  MoveL 4411 to (296.71, 215.61, -10) mm, rotated rx -180 ry 0 rz 180 deg; joints [-8.145, -42.25, 106.462, 170.968, 64.491, -176.084]
  MoveL 4412 to (298.79, 218.64, -10) mm, rotated rx 180 ry 0 rz 180 deg; joints [-8.247, -42.193, 106.293, 170.847, 64.387, -176.016]
  MoveL 4413 to (300.68, 221.8, -10) mm, rotated rx 180 ry 0 rz 180 deg; joints [-8.354, -42.14, 106.135, 170.72, 64.292, -175.946]
  MoveL 4414 to (302.37, 225.07, -10) mm, rotated rx -180 ry 0 rz -180 deg; joints [-8.466, -42.091, 105.99, 170.589, 64.205, -175.874]
  MoveL 4415 to (303.85, 228.44, -10) mm, rotated rx -180 ry 0 rz 180 deg; joints [-8.583, -42.046, 105.857, 170.452, 64.127, -175.802]
  MoveL 4416 to (305.1, 231.9, -10) mm, rotated rx -180 ry 0 rz -180 deg; joints [-8.704, -42.005, 105.737, 170.312, 64.058, -175.729]
  MoveL 4417 to (306.14, 235.43, -10) mm, rotated rx 180 ry 0 rz 180 deg; joints [-8.828, -41.969, 105.631, 170.168, 63.998, -175.655]
  MoveL 4418 to (306.95, 239.02, -10) mm, rotated rx 180 ry 0 rz -180 deg; joints [-8.956, -41.937, 105.539, 170.021, 63.948, -175.581]
  MoveL 4419 to (307.53, 242.66, -10) mm, rotated rx -180 ry 0 rz 180 deg; joints [-9.087, -41.911, 105.461, 169.872, 63.908, -175.508]
  MoveL 4420 to (307.88, 246.32, -10) mm, rotated rx -180 ry 0 rz -180 deg; joints [-9.219, -41.889, 105.398, 169.721, 63.877, -175.435]
  MoveL 4421 to (308, 250, -10) mm, rotated rx 180 ry 0 rz 180 deg; joints [-9.354, -41.873, 105.35, 169.569, 63.857, -175.363]
  MoveL 4422 to (296, 250, -10) mm, rotated rx 180 ry 0 rz 180 deg; joints [-9.427, -42.146, 106.154, 169.534, 64.384, -175.434]
  MoveL 4423 to (295.91, 252.92, -10) mm, rotated rx -180 ry 0 rz 180 deg; joints [-9.536, -42.137, 106.127, 169.413, 64.376, -175.379]
  MoveL 4424 to (295.63, 255.82, -10) mm, rotated rx -180 ry 0 rz 180 deg; joints [-9.645, -42.132, 106.113, 169.291, 64.375, -175.324]
  MoveL 4425 to (295.17, 258.71, -10) mm, rotated rx -180 ry 0 rz -180 deg; joints [-9.755, -42.132, 106.111, 169.17, 64.383, -175.272]
  MoveL 4426 to (294.53, 261.55, -10) mm, rotated rx -180 ry 0 rz 180 deg; joints [-9.864, -42.135, 106.121, 169.05, 64.399, -175.221]
  MoveL 4427 to (293.7, 264.35, -10) mm, rotated rx 180 ry 0 rz 180 deg; joints [-9.973, -42.142, 106.143, 168.931, 64.422, -175.172]
  MoveL 4428 to (292.7, 267.1, -10) mm, rotated rx 180 ry 0 rz 180 deg; joints [-10.081, -42.154, 106.177, 168.814, 64.453, -175.125]
  MoveL 4429 to (291.53, 269.77, -10) mm, rotated rx 180 ry 0 rz 180 deg; joints [-10.187, -42.17, 106.223, 168.699, 64.493, -175.081]
  MoveL 4430 to (290.2, 272.37, -10) mm, rotated rx -180 ry 0 rz -180 deg; joints [-10.292, -42.189, 106.281, 168.587, 64.539, -175.04]
  MoveL 4431 to (288.7, 274.87, -10) mm, rotated rx 180 ry 0 rz 180 deg; joints [-10.395, -42.213, 106.351, 168.478, 64.593, -175.001]
  MoveL 4432 to (287.04, 277.27, -10) mm, rotated rx 180 ry 0 rz 180 deg; joints [-10.495, -42.24, 106.431, 168.372, 64.654, -174.966]
  MoveL 4433 to (285.24, 279.57, -10) mm, rotated rx 180 ry 0 rz 180 deg; joints [-10.593, -42.271, 106.523, 168.271, 64.722, -174.934]
  MoveL 4434 to (283.29, 281.74, -10) mm, rotated rx 180 ry 0 rz -180 deg; joints [-10.687, -42.305, 106.625, 168.174, 64.797, -174.905]
  MoveL 4435 to (281.21, 283.79, -10) mm, rotated rx -180 ry 0 rz -180 deg; joints [-10.777, -42.342, 106.737, 168.081, 64.878, -174.879]
  MoveL 4436 to (279.01, 285.7, -10) mm, rotated rx 180 ry 0 rz -180 deg; joints [-10.864, -42.383, 106.859, 167.994, 64.965, -174.857]
  MoveL 4437 to (276.68, 287.47, -10) mm, rotated rx 180 ry 0 rz 180 deg; joints [-10.946, -42.427, 106.99, 167.912, 65.058, -174.839]
  MoveL 4438 to (274.25, 289.09, -10) mm, rotated rx -180 ry 0 rz -180 deg; joints [-11.024, -42.474, 107.13, 167.836, 65.156, -174.825]
  MoveL 4439 to (271.72, 290.55, -10) mm, rotated rx 180 ry 0 rz -180 deg; joints [-11.096, -42.523, 107.278, 167.766, 65.259, -174.815]
  MoveL 4440 to (269.11, 291.84, -10) mm, rotated rx 180 ry 0 rz -180 deg; joints [-11.164, -42.575, 107.433, 167.702, 65.366, -174.808]
  MoveL 4441 to (266.42, 292.97, -10) mm, rotated rx -180 ry 0 rz -180 deg; joints [-11.226, -42.629, 107.596, 167.644, 65.478, -174.805]
  MoveL 4442 to (263.66, 293.93, -10) mm, rotated rx -180 ry 0 rz -180 deg; joints [-11.282, -42.685, 107.765, 167.594, 65.594, -174.806]
  MoveL 4443 to (260.84, 294.7, -10) mm, rotated rx -180 ry 0 rz -180 deg; joints [-11.332, -42.742, 107.939, 167.551, 65.712, -174.811]
  MoveL 4444 to (257.99, 295.3, -10) mm, rotated rx -180 ry 0 rz 180 deg; joints [-11.376, -42.801, 108.119, 167.514, 65.834, -174.82]
  MoveL 4445 to (255.1, 295.72, -10) mm, rotated rx -180 ry 0 rz -180 deg; joints [-11.414, -42.861, 108.303, 167.485, 65.958, -174.833]
  MoveL 4446 to (252.19, 295.95, -10) mm, rotated rx 180 ry 0 rz -180 deg; joints [-11.444, -42.923, 108.49, 167.464, 66.084, -174.849]
  MoveL 4447 to (249.27, 295.99, -10) mm, rotated rx 180 ry 0 rz 180 deg; joints [-11.468, -42.985, 108.68, 167.45, 66.211, -174.869]
  MoveL 4448 to (246.35, 295.86, -10) mm, rotated rx 180 ry 0 rz -180 deg; joints [-11.486, -43.047, 108.872, 167.444, 66.339, -174.892]
  MoveL 4449 to (243.45, 295.53, -10) mm, rotated rx 180 ry 0 rz -180 deg; joints [-11.496, -43.11, 109.065, 167.445, 66.467, -174.919]
  MoveL 4450 to (240.58, 295.02, -10) mm, rotated rx -180 ry 0 rz -180 deg; joints [-11.499, -43.172, 109.259, 167.454, 66.596, -174.949]
  MoveL 4451 to (237.74, 294.34, -10) mm, rotated rx 180 ry 0 rz 180 deg; joints [-11.494, -43.234, 109.452, 167.471, 66.723, -174.981]
  MoveL 4452 to (234.95, 293.47, -10) mm, rotated rx -180 ry 0 rz -180 deg; joints [-11.483, -43.296, 109.645, 167.496, 66.85, -175.017]
  MoveL 4453 to (232.23, 292.43, -10) mm, rotated rx 180 ry 0 rz -180 deg; joints [-11.464, -43.357, 109.835, 167.528, 66.975, -175.056]
  MoveL 4454 to (229.57, 291.22, -10) mm, rotated rx -180 ry 0 rz 180 deg; joints [-11.439, -43.417, 110.023, 167.568, 67.098, -175.096]
  MoveL 4455 to (227, 289.84, -10) mm, rotated rx -180 ry 0 rz -180 deg; joints [-11.406, -43.475, 110.207, 167.615, 67.218, -175.14]
  MoveL 4456 to (224.52, 288.3, -10) mm, rotated rx 180 ry 0 rz 180 deg; joints [-11.366, -43.532, 110.388, 167.669, 67.335, -175.185]
  MoveL 4457 to (222.14, 286.6, -10) mm, rotated rx -180 ry 0 rz -180 deg; joints [-11.319, -43.588, 110.563, 167.73, 67.448, -175.232]
  MoveL 4458 to (219.88, 284.76, -10) mm, rotated rx 180 ry 0 rz -180 deg; joints [-11.266, -43.641, 110.733, 167.798, 67.558, -175.281]
  MoveL 4459 to (217.73, 282.78, -10) mm, rotated rx -180 ry 0 rz -180 deg; joints [-11.206, -43.692, 110.897, 167.872, 67.663, -175.331]
  MoveL 4460 to (215.72, 280.67, -10) mm, rotated rx 180 ry 0 rz 180 deg; joints [-11.139, -43.741, 111.053, 167.953, 67.762, -175.382]
  MoveL 4461 to (213.84, 278.44, -10) mm, rotated rx 180 ry 0 rz -180 deg; joints [-11.067, -43.788, 111.202, 168.039, 67.857, -175.435]
  MoveL 4462 to (212.11, 276.08, -10) mm, rotated rx -180 ry 0 rz -180 deg; joints [-10.989, -43.832, 111.343, 168.131, 67.946, -175.488]
  MoveL 4463 to (210.53, 273.63, -10) mm, rotated rx -180 ry 0 rz -180 deg; joints [-10.905, -43.873, 111.475, 168.229, 68.028, -175.542]
  MoveL 4464 to (209.11, 271.08, -10) mm, rotated rx 180 ry 0 rz 180 deg; joints [-10.817, -43.91, 111.598, 168.331, 68.104, -175.596]
  MoveL 4465 to (207.86, 268.44, -10) mm, rotated rx -180 ry 0 rz -180 deg; joints [-10.723, -43.945, 111.71, 168.438, 68.174, -175.65]
  MoveL 4466 to (206.77, 265.73, -10) mm, rotated rx 180 ry 0 rz -180 deg; joints [-10.625, -43.977, 111.813, 168.549, 68.236, -175.705]
  MoveL 4467 to (205.86, 262.96, -10) mm, rotated rx 180 ry 0 rz -180 deg; joints [-10.523, -44.005, 111.905, 168.663, 68.29, -175.759]
  MoveL 4468 to (205.13, 260.13, -10) mm, rotated rx 180 ry 0 rz -180 deg; joints [-10.418, -44.03, 111.985, 168.78, 68.337, -175.812]
  MoveL 4469 to (204.58, 257.27, -10) mm, rotated rx 180 ry 0 rz 180 deg; joints [-10.31, -44.051, 112.054, 168.9, 68.377, -175.865]
  MoveL 4470 to (204.21, 254.37, -10) mm, rotated rx -180 ry 0 rz 180 deg; joints [-10.199, -44.068, 112.112, 169.022, 68.408, -175.917]
  MoveL 4471 to (204.02, 251.46, -10) mm, rotated rx 180 ry 0 rz 180 deg; joints [-10.086, -44.082, 112.157, 169.146, 68.431, -175.968]
  MoveL 4472 to (204.02, 248.54, -10) mm, rotated rx 180 ry 0 rz 180 deg; joints [-9.971, -44.092, 112.19, 169.271, 68.445, -176.018]
  MoveL 4473 to (204.21, 245.63, -10) mm, rotated rx 180 ry 0 rz -180 deg; joints [-9.855, -44.099, 112.211, 169.396, 68.451, -176.066]
  MoveL 4474 to (204.58, 242.73, -10) mm, rotated rx 180 ry 0 rz -180 deg; joints [-9.739, -44.101, 112.219, 169.521, 68.449, -176.113]
  MoveL 4475 to (205.13, 239.87, -10) mm, rotated rx 180 ry 0 rz -180 deg; joints [-9.622, -44.1, 112.215, 169.646, 68.439, -176.159]
  MoveL 4476 to (205.86, 237.04, -10) mm, rotated rx 180 ry 0 rz 180 deg; joints [-9.506, -44.095, 112.199, 169.77, 68.42, -176.202]
  MoveL 4477 to (206.77, 234.27, -10) mm, rotated rx -180 ry 0 rz 180 deg; joints [-9.391, -44.086, 112.17, 169.892, 68.392, -176.244]
  MoveL 4478 to (207.86, 231.56, -10) mm, rotated rx -180 ry 0 rz -180 deg; joints [-9.277, -44.074, 112.129, 170.012, 68.357, -176.284]
  MoveL 4479 to (209.11, 228.92, -10) mm, rotated rx 180 ry 0 rz 180 deg; joints [-9.166, -44.057, 112.075, 170.13, 68.313, -176.321]
  MoveL 4480 to (210.53, 226.37, -10) mm, rotated rx 180 ry 0 rz -180 deg; joints [-9.056, -44.037, 112.01, 170.244, 68.262, -176.356]
  MoveL 4481 to (212.11, 223.92, -10) mm, rotated rx -180 ry 0 rz 180 deg; joints [-8.95, -44.014, 111.934, 170.355, 68.202, -176.389]
  MoveL 4482 to (213.84, 221.56, -10) mm, rotated rx 180 ry 0 rz 180 deg; joints [-8.847, -43.987, 111.846, 170.461, 68.136, -176.419]
  MoveL 4483 to (215.72, 219.33, -10) mm, rotated rx -180 ry 0 rz 180 deg; joints [-8.747, -43.957, 111.747, 170.564, 68.062, -176.447]
  MoveL 4484 to (217.73, 217.22, -10) mm, rotated rx -180 ry 0 rz 180 deg; joints [-8.652, -43.923, 111.638, 170.661, 67.982, -176.472]
  MoveL 4485 to (219.88, 215.24, -10) mm, rotated rx 180 ry 0 rz 180 deg; joints [-8.562, -43.886, 111.518, 170.753, 67.895, -176.494]
  MoveL 4486 to (222.14, 213.4, -10) mm, rotated rx 180 ry 0 rz -180 deg; joints [-8.477, -43.846, 111.39, 170.839, 67.802, -176.513]
  MoveL 4487 to (224.52, 211.7, -10) mm, rotated rx 180 ry 0 rz -180 deg; joints [-8.397, -43.803, 111.252, 170.919, 67.703, -176.53]
  MoveL 4488 to (227, 210.16, -10) mm, rotated rx -180 ry 0 rz 180 deg; joints [-8.322, -43.758, 111.106, 170.993, 67.599, -176.543]
  MoveL 4489 to (229.57, 208.78, -10) mm, rotated rx 180 ry 0 rz -180 deg; joints [-8.254, -43.71, 110.952, 171.06, 67.491, -176.554]
  MoveL 4490 to (232.23, 207.57, -10) mm, rotated rx 180 ry 0 rz -180 deg; joints [-8.192, -43.659, 110.79, 171.12, 67.378, -176.561]
  MoveL 4491 to (234.95, 206.53, -10) mm, rotated rx 180 ry 0 rz 180 deg; joints [-8.136, -43.606, 110.623, 171.173, 67.261, -176.565]
  MoveL 4492 to (237.74, 205.66, -10) mm, rotated rx -180 ry 0 rz -180 deg; joints [-8.087, -43.552, 110.449, 171.219, 67.14, -176.566]
  MoveL 4493 to (240.58, 204.98, -10) mm, rotated rx -180 ry 0 rz -180 deg; joints [-8.045, -43.495, 110.27, 171.257, 67.017, -176.563]
  MoveL 4494 to (243.45, 204.47, -10) mm, rotated rx 180 ry 0 rz 180 deg; joints [-8.009, -43.437, 110.087, 171.287, 66.891, -176.558]
  MoveL 4495 to (246.35, 204.14, -10) mm, rotated rx -180 ry 0 rz 180 deg; joints [-7.981, -43.378, 109.9, 171.309, 66.763, -176.549]
  MoveL 4496 to (249.27, 204.01, -10) mm, rotated rx -180 ry 0 rz -180 deg; joints [-7.96, -43.317, 109.711, 171.324, 66.635, -176.537]
  MoveL 4497 to (252.19, 204.05, -10) mm, rotated rx 180 ry 0 rz -180 deg; joints [-7.946, -43.256, 109.519, 171.33, 66.505, -176.521]
  MoveL 4498 to (255.1, 204.28, -10) mm, rotated rx -180 ry 0 rz -180 deg; joints [-7.939, -43.194, 109.326, 171.329, 66.375, -176.503]
  MoveL 4499 to (257.99, 204.7, -10) mm, rotated rx 180 ry 0 rz 180 deg; joints [-7.94, -43.131, 109.132, 171.32, 66.245, -176.481]
  MoveL 4500 to (260.84, 205.3, -10) mm, rotated rx 180 ry 0 rz 180 deg; joints [-7.947, -43.069, 108.938, 171.303, 66.116, -176.456]
  MoveL 4501 to (263.66, 206.07, -10) mm, rotated rx -180 ry 0 rz -180 deg; joints [-7.962, -43.006, 108.746, 171.278, 65.989, -176.428]
  MoveL 4502 to (266.42, 207.03, -10) mm, rotated rx -180 ry 0 rz -180 deg; joints [-7.984, -42.944, 108.555, 171.246, 65.863, -176.397]
  MoveL 4503 to (269.11, 208.16, -10) mm, rotated rx 180 ry 0 rz 180 deg; joints [-8.012, -42.882, 108.367, 171.206, 65.739, -176.363]
  MoveL 4504 to (271.72, 209.45, -10) mm, rotated rx -180 ry 0 rz -180 deg; joints [-8.047, -42.822, 108.182, 171.159, 65.619, -176.326]
  MoveL 4505 to (274.25, 210.91, -10) mm, rotated rx -180 ry 0 rz -180 deg; joints [-8.089, -42.762, 108.001, 171.104, 65.501, -176.286]
  MoveL 4506 to (276.68, 212.53, -10) mm, rotated rx 180 ry 0 rz -180 deg; joints [-8.137, -42.704, 107.824, 171.043, 65.387, -176.244]
  MoveL 4507 to (279.01, 214.3, -10) mm, rotated rx 180 ry 0 rz -180 deg; joints [-8.191, -42.648, 107.654, 170.976, 65.278, -176.2]
  MoveL 4508 to (281.21, 216.21, -10) mm, rotated rx -180 ry 0 rz 180 deg; joints [-8.251, -42.593, 107.489, 170.902, 65.173, -176.153]
  MoveL 4509 to (283.29, 218.26, -10) mm, rotated rx 180 ry 0 rz 180 deg; joints [-8.317, -42.541, 107.331, 170.822, 65.073, -176.104]
  MoveL 4510 to (285.24, 220.43, -10) mm, rotated rx 180 ry 0 rz -180 deg; joints [-8.388, -42.491, 107.18, 170.736, 64.979, -176.054]
  MoveL 4511 to (287.04, 222.73, -10) mm, rotated rx 180 ry 0 rz 180 deg; joints [-8.464, -42.443, 107.037, 170.645, 64.89, -176.001]
  MoveL 4512 to (288.7, 225.13, -10) mm, rotated rx 180 ry 0 rz -180 deg; joints [-8.545, -42.398, 106.903, 170.549, 64.808, -175.947]
  MoveL 4513 to (290.2, 227.64, -10) mm, rotated rx -180 ry 0 rz -180 deg; joints [-8.63, -42.356, 106.778, 170.449, 64.732, -175.892]
  MoveL 4514 to (291.53, 230.23, -10) mm, rotated rx 180 ry 0 rz 180 deg; joints [-8.719, -42.317, 106.662, 170.345, 64.663, -175.836]
  MoveL 4515 to (292.7, 232.9, -10) mm, rotated rx 180 ry 0 rz 180 deg; joints [-8.812, -42.282, 106.557, 170.236, 64.6, -175.779]
  MoveL 4516 to (293.7, 235.65, -10) mm, rotated rx -180 ry 0 rz -180 deg; joints [-8.908, -42.25, 106.462, 170.125, 64.545, -175.721]
  MoveL 4517 to (294.53, 238.45, -10) mm, rotated rx -180 ry 0 rz -180 deg; joints [-9.007, -42.222, 106.377, 170.011, 64.497, -175.663]
  MoveL 4518 to (295.17, 241.29, -10) mm, rotated rx -180 ry 0 rz -180 deg; joints [-9.109, -42.197, 106.304, 169.894, 64.457, -175.605]
  MoveL 4519 to (295.63, 244.18, -10) mm, rotated rx 180 ry 0 rz 180 deg; joints [-9.214, -42.176, 106.242, 169.775, 64.425, -175.548]
  MoveL 4520 to (295.91, 247.08, -10) mm, rotated rx -180 ry 0 rz -180 deg; joints [-9.32, -42.159, 106.192, 169.655, 64.401, -175.49]
  MoveL 4521 to (296, 250, -10) mm, rotated rx 180 ry 0 rz 180 deg; joints [-9.427, -42.146, 106.154, 169.534, 64.384, -175.434]
  MoveL 4522 to (284, 250, -10) mm, rotated rx -180 ry 0 rz 180 deg; joints [-9.502, -42.415, 106.953, 169.498, 64.912, -175.506]
  MoveL 4523 to (283.93, 252.16, -10) mm, rotated rx 180 ry 0 rz -180 deg; joints [-9.582, -42.408, 106.933, 169.408, 64.905, -175.465]
  MoveL 4524 to (283.73, 254.3, -10) mm, rotated rx -180 ry 0 rz 180 deg; joints [-9.664, -42.405, 106.923, 169.318, 64.905, -175.426]
  MoveL 4525 to (283.39, 256.43, -10) mm, rotated rx 180 ry 0 rz -180 deg; joints [-9.745, -42.404, 106.921, 169.228, 64.91, -175.388]
  MoveL 4526 to (282.91, 258.54, -10) mm, rotated rx 180 ry 0 rz 180 deg; joints [-9.827, -42.407, 106.929, 169.139, 64.922, -175.351]
  MoveL 4527 to (282.3, 260.61, -10) mm, rotated rx 180 ry 0 rz -180 deg; joints [-9.908, -42.412, 106.945, 169.05, 64.939, -175.315]
  MoveL 4528 to (281.56, 262.64, -10) mm, rotated rx 180 ry 0 rz 180 deg; joints [-9.988, -42.421, 106.971, 168.963, 64.962, -175.281]
  MoveL 4529 to (280.7, 264.61, -10) mm, rotated rx 180 ry 0 rz 180 deg; joints [-10.068, -42.432, 107.005, 168.878, 64.991, -175.249]
  MoveL 4530 to (279.71, 266.53, -10) mm, rotated rx 180 ry 0 rz 180 deg; joints [-10.146, -42.446, 107.048, 168.795, 65.026, -175.219]
  MoveL 4531 to (278.6, 268.38, -10) mm, rotated rx 180 ry 0 rz 180 deg; joints [-10.222, -42.464, 107.099, 168.714, 65.066, -175.191]
  MoveL 4532 to (277.38, 270.16, -10) mm, rotated rx -180 ry 0 rz -180 deg; joints [-10.297, -42.483, 107.159, 168.636, 65.111, -175.165]
  MoveL 4533 to (276.05, 271.85, -10) mm, rotated rx 180 ry 0 rz -180 deg; joints [-10.369, -42.506, 107.226, 168.56, 65.161, -175.141]
  MoveL 4534 to (274.61, 273.46, -10) mm, rotated rx 180 ry 0 rz 180 deg; joints [-10.439, -42.531, 107.302, 168.488, 65.217, -175.12]
  MoveL 4535 to (273.07, 274.98, -10) mm, rotated rx 180 ry 0 rz 180 deg; joints [-10.506, -42.559, 107.385, 168.42, 65.277, -175.102]
  MoveL 4536 to (271.44, 276.39, -10) mm, rotated rx -180 ry 0 rz 180 deg; joints [-10.57, -42.589, 107.475, 168.355, 65.341, -175.086]
  MoveL 4537 to (269.72, 277.7, -10) mm, rotated rx 180 ry 0 rz 180 deg; joints [-10.631, -42.621, 107.572, 168.294, 65.41, -175.072]
  MoveL 4538 to (267.93, 278.89, -10) mm, rotated rx 180 ry 0 rz 180 deg; joints [-10.688, -42.655, 107.676, 168.238, 65.483, -175.062]
  MoveL 4539 to (266.06, 279.97, -10) mm, rotated rx 180 ry 0 rz 180 deg; joints [-10.742, -42.691, 107.786, 168.186, 65.56, -175.054]
  MoveL 4540 to (264.12, 280.93, -10) mm, rotated rx 180 ry 0 rz -180 deg; joints [-10.792, -42.729, 107.901, 168.139, 65.639, -175.049]
  MoveL 4541 to (262.13, 281.76, -10) mm, rotated rx 180 ry 0 rz 180 deg; joints [-10.837, -42.769, 108.021, 168.097, 65.722, -175.047]
  MoveL 4542 to (260.1, 282.47, -10) mm, rotated rx 180 ry 0 rz -180 deg; joints [-10.879, -42.81, 108.146, 168.059, 65.808, -175.047]
  MoveL 4543 to (258.02, 283.04, -10) mm, rotated rx -180 ry 0 rz -180 deg; joints [-10.915, -42.852, 108.275, 168.027, 65.896, -175.05]
  MoveL 4544 to (255.9, 283.48, -10) mm, rotated rx 180 ry 0 rz -180 deg; joints [-10.947, -42.896, 108.408, 168.001, 65.986, -175.056]
  MoveL 4545 to (253.77, 283.79, -10) mm, rotated rx -180 ry 0 rz 180 deg; joints [-10.974, -42.94, 108.544, 167.98, 66.078, -175.065]
  MoveL 4546 to (251.62, 283.96, -10) mm, rotated rx 180 ry 0 rz -180 deg; joints [-10.997, -42.985, 108.683, 167.964, 66.171, -175.077]
  MoveL 4547 to (249.46, 284, -10) mm, rotated rx 180 ry 0 rz -180 deg; joints [-11.014, -43.031, 108.823, 167.954, 66.266, -175.091]
  MoveL 4548 to (247.31, 283.89, -10) mm, rotated rx -180 ry 0 rz -180 deg; joints [-11.026, -43.077, 108.965, 167.95, 66.36, -175.107]
  MoveL 4549 to (245.16, 283.65, -10) mm, rotated rx -180 ry 0 rz 180 deg; joints [-11.033, -43.123, 109.108, 167.951, 66.456, -175.127]
  MoveL 4550 to (243.04, 283.28, -10) mm, rotated rx 180 ry 0 rz 180 deg; joints [-11.034, -43.17, 109.251, 167.958, 66.551, -175.148]
  MoveL 4551 to (240.94, 282.77, -10) mm, rotated rx -180 ry 0 rz 180 deg; joints [-11.03, -43.216, 109.394, 167.971, 66.645, -175.172]
  MoveL 4552 to (238.88, 282.13, -10) mm, rotated rx 180 ry 0 rz -180 deg; joints [-11.021, -43.261, 109.536, 167.99, 66.739, -175.197]
  MoveL 4553 to (236.86, 281.36, -10) mm, rotated rx -180 ry 0 rz -180 deg; joints [-11.007, -43.306, 109.677, 168.014, 66.831, -175.225]
  MoveL 4554 to (234.9, 280.46, -10) mm, rotated rx -180 ry 0 rz -180 deg; joints [-10.987, -43.351, 109.816, 168.044, 66.922, -175.255]
  MoveL 4555 to (233, 279.44, -10) mm, rotated rx 180 ry 0 rz -180 deg; joints [-10.962, -43.394, 109.952, 168.079, 67.01, -175.286]
  MoveL 4556 to (231.17, 278.31, -10) mm, rotated rx 180 ry 0 rz -180 deg; joints [-10.932, -43.437, 110.085, 168.119, 67.097, -175.319]
  MoveL 4557 to (229.41, 277.06, -10) mm, rotated rx 180 ry 0 rz 180 deg; joints [-10.897, -43.478, 110.215, 168.165, 67.18, -175.354]
  MoveL 4558 to (227.73, 275.7, -10) mm, rotated rx -180 ry 0 rz 180 deg; joints [-10.857, -43.517, 110.34, 168.215, 67.261, -175.389]
  MoveL 4559 to (226.15, 274.23, -10) mm, rotated rx 180 ry 0 rz 180 deg; joints [-10.813, -43.555, 110.461, 168.27, 67.338, -175.426]
  MoveL 4560 to (224.66, 272.67, -10) mm, rotated rx 180 ry 0 rz -180 deg; joints [-10.763, -43.592, 110.576, 168.33, 67.412, -175.464]
  MoveL 4561 to (223.27, 271.02, -10) mm, rotated rx -180 ry 0 rz -180 deg; joints [-10.71, -43.626, 110.686, 168.394, 67.481, -175.503]
  MoveL 4562 to (221.99, 269.28, -10) mm, rotated rx 180 ry 0 rz -180 deg; joints [-10.652, -43.659, 110.79, 168.463, 67.547, -175.542]
  MoveL 4563 to (220.83, 267.46, -10) mm, rotated rx -180 ry 0 rz 180 deg; joints [-10.59, -43.69, 110.887, 168.535, 67.607, -175.582]
  MoveL 4564 to (219.78, 265.58, -10) mm, rotated rx -180 ry 0 rz -180 deg; joints [-10.525, -43.718, 110.978, 168.61, 67.663, -175.622]
  MoveL 4565 to (218.85, 263.63, -10) mm, rotated rx 180 ry 0 rz 180 deg; joints [-10.456, -43.744, 111.061, 168.689, 67.714, -175.662]
  MoveL 4566 to (218.05, 261.63, -10) mm, rotated rx -180 ry 0 rz -180 deg; joints [-10.384, -43.767, 111.136, 168.771, 67.76, -175.703]
  MoveL 4567 to (217.38, 259.58, -10) mm, rotated rx -180 ry 0 rz -180 deg; joints [-10.309, -43.788, 111.204, 168.855, 67.8, -175.743]
  MoveL 4568 to (216.84, 257.49, -10) mm, rotated rx -180 ry 0 rz -180 deg; joints [-10.232, -43.807, 111.263, 168.942, 67.834, -175.783]
  MoveL 4569 to (216.43, 255.37, -10) mm, rotated rx 180 ry 0 rz 180 deg; joints [-10.152, -43.823, 111.314, 169.03, 67.863, -175.822]
  MoveL 4570 to (216.15, 253.23, -10) mm, rotated rx 180 ry 0 rz -180 deg; joints [-10.071, -43.836, 111.356, 169.12, 67.885, -175.861]
  MoveL 4571 to (216.02, 251.08, -10) mm, rotated rx -180 ry 0 rz -180 deg; joints [-9.988, -43.846, 111.39, 169.211, 67.902, -175.9]
  MoveL 4572 to (216.02, 248.92, -10) mm, rotated rx -180 ry 0 rz 180 deg; joints [-9.904, -43.854, 111.414, 169.303, 67.913, -175.937]
  MoveL 4573 to (216.15, 246.77, -10) mm, rotated rx -180 ry 0 rz 180 deg; joints [-9.819, -43.858, 111.429, 169.395, 67.917, -175.974]
  MoveL 4574 to (216.43, 244.63, -10) mm, rotated rx 180 ry 0 rz -180 deg; joints [-9.733, -43.86, 111.436, 169.487, 67.915, -176.009]
  MoveL 4575 to (216.84, 242.51, -10) mm, rotated rx -180 ry 0 rz 180 deg; joints [-9.648, -43.859, 111.433, 169.579, 67.907, -176.043]
  MoveL 4576 to (217.38, 240.42, -10) mm, rotated rx -180 ry 0 rz -180 deg; joints [-9.563, -43.856, 111.42, 169.67, 67.893, -176.076]
  MoveL 4577 to (218.05, 238.37, -10) mm, rotated rx -180 ry 0 rz -180 deg; joints [-9.478, -43.849, 111.399, 169.76, 67.873, -176.107]
  MoveL 4578 to (218.85, 236.37, -10) mm, rotated rx 180 ry 0 rz 180 deg; joints [-9.395, -43.84, 111.369, 169.848, 67.847, -176.137]
  MoveL 4579 to (219.78, 234.42, -10) mm, rotated rx 180 ry 0 rz -180 deg; joints [-9.313, -43.827, 111.33, 169.935, 67.815, -176.166]
  MoveL 4580 to (220.83, 232.53, -10) mm, rotated rx -180 ry 0 rz 180 deg; joints [-9.233, -43.813, 111.282, 170.019, 67.777, -176.192]
  MoveL 4581 to (221.99, 230.72, -10) mm, rotated rx 180 ry 0 rz -180 deg; joints [-9.155, -43.795, 111.225, 170.101, 67.733, -176.217]
  MoveL 4582 to (223.27, 228.98, -10) mm, rotated rx -180 ry 0 rz 180 deg; joints [-9.079, -43.775, 111.16, 170.179, 67.684, -176.239]
  MoveL 4583 to (224.66, 227.33, -10) mm, rotated rx -180 ry 0 rz 180 deg; joints [-9.006, -43.752, 111.088, 170.254, 67.63, -176.26]
  MoveL 4584 to (226.15, 225.77, -10) mm, rotated rx -180 ry 0 rz 180 deg; joints [-8.936, -43.727, 111.007, 170.326, 67.571, -176.279]
  MoveL 4585 to (227.73, 224.3, -10) mm, rotated rx -180 ry 0 rz 180 deg; joints [-8.869, -43.7, 110.919, 170.394, 67.507, -176.295]
  MoveL 4586 to (229.41, 222.94, -10) mm, rotated rx 180 ry 0 rz 180 deg; joints [-8.806, -43.67, 110.824, 170.458, 67.439, -176.31]
  MoveL 4587 to (231.17, 221.69, -10) mm, rotated rx -180 ry 0 rz 180 deg; joints [-8.747, -43.638, 110.723, 170.517, 67.366, -176.322]
  MoveL 4588 to (233, 220.56, -10) mm, rotated rx 180 ry 0 rz -180 deg; joints [-8.692, -43.604, 110.615, 170.571, 67.29, -176.332]
  MoveL 4589 to (234.9, 219.54, -10) mm, rotated rx 180 ry 0 rz -180 deg; joints [-8.641, -43.568, 110.501, 170.621, 67.21, -176.339]
  MoveL 4590 to (236.86, 218.64, -10) mm, rotated rx -180 ry 0 rz 180 deg; joints [-8.595, -43.531, 110.382, 170.665, 67.126, -176.344]
  MoveL 4591 to (238.88, 217.87, -10) mm, rotated rx -180 ry 0 rz 180 deg; joints [-8.553, -43.491, 110.258, 170.705, 67.04, -176.347]
  MoveL 4592 to (240.94, 217.23, -10) mm, rotated rx 180 ry 0 rz 180 deg; joints [-8.517, -43.451, 110.13, 170.738, 66.952, -176.347]
  MoveL 4593 to (243.04, 216.72, -10) mm, rotated rx 180 ry 0 rz 180 deg; joints [-8.485, -43.409, 109.998, 170.767, 66.861, -176.345]
  MoveL 4594 to (245.16, 216.35, -10) mm, rotated rx 180 ry 0 rz 180 deg; joints [-8.458, -43.366, 109.863, 170.789, 66.768, -176.34]
  MoveL 4595 to (247.31, 216.11, -10) mm, rotated rx 180 ry 0 rz 180 deg; joints [-8.437, -43.322, 109.725, 170.806, 66.674, -176.333]
  MoveL 4596 to (249.46, 216, -10) mm, rotated rx 180 ry 0 rz -180 deg; joints [-8.421, -43.277, 109.585, 170.817, 66.579, -176.323]
  MoveL 4597 to (251.62, 216.04, -10) mm, rotated rx -180 ry 0 rz -180 deg; joints [-8.41, -43.231, 109.443, 170.822, 66.483, -176.311]
  MoveL 4598 to (253.77, 216.21, -10) mm, rotated rx 180 ry 0 rz -180 deg; joints [-8.404, -43.186, 109.301, 170.822, 66.387, -176.297]
  MoveL 4599 to (255.9, 216.52, -10) mm, rotated rx -180 ry 0 rz 180 deg; joints [-8.404, -43.139, 109.157, 170.815, 66.291, -176.28]
  MoveL 4600 to (258.02, 216.96, -10) mm, rotated rx 180 ry 0 rz -180 deg; joints [-8.409, -43.093, 109.014, 170.803, 66.196, -176.261]
  MoveL 4601 to (260.1, 217.53, -10) mm, rotated rx 180 ry 0 rz 180 deg; joints [-8.419, -43.047, 108.872, 170.785, 66.102, -176.24]
  MoveL 4602 to (262.13, 218.24, -10) mm, rotated rx 180 ry 0 rz 180 deg; joints [-8.434, -43.001, 108.731, 170.762, 66.009, -176.216]
  MoveL 4603 to (264.12, 219.07, -10) mm, rotated rx -180 ry 0 rz 180 deg; joints [-8.455, -42.956, 108.592, 170.732, 65.917, -176.191]
  MoveL 4604 to (266.06, 220.03, -10) mm, rotated rx -180 ry 0 rz 180 deg; joints [-8.48, -42.911, 108.455, 170.698, 65.828, -176.163]
  MoveL 4605 to (267.93, 221.11, -10) mm, rotated rx 180 ry 0 rz 180 deg; joints [-8.51, -42.867, 108.321, 170.658, 65.741, -176.133]
  MoveL 4606 to (269.72, 222.3, -10) mm, rotated rx -180 ry 0 rz -180 deg; joints [-8.546, -42.825, 108.19, 170.613, 65.657, -176.102]
  MoveL 4607 to (271.44, 223.61, -10) mm, rotated rx -180 ry 0 rz -180 deg; joints [-8.585, -42.783, 108.064, 170.564, 65.576, -176.069]
  MoveL 4608 to (273.07, 225.02, -10) mm, rotated rx 180 ry 0 rz 180 deg; joints [-8.629, -42.743, 107.942, 170.509, 65.498, -176.034]
  MoveL 4609 to (274.61, 226.54, -10) mm, rotated rx 180 ry 0 rz -180 deg; joints [-8.678, -42.704, 107.825, 170.45, 65.424, -175.998]
  MoveL 4610 to (276.05, 228.15, -10) mm, rotated rx -180 ry 0 rz -180 deg; joints [-8.73, -42.668, 107.713, 170.387, 65.354, -175.96]
  MoveL 4611 to (277.38, 229.84, -10) mm, rotated rx 180 ry 0 rz -180 deg; joints [-8.786, -42.633, 107.608, 170.32, 65.288, -175.921]
  MoveL 4612 to (278.6, 231.62, -10) mm, rotated rx -180 ry 0 rz -180 deg; joints [-8.846, -42.6, 107.508, 170.249, 65.227, -175.882]
  MoveL 4613 to (279.71, 233.47, -10) mm, rotated rx -180 ry 0 rz -180 deg; joints [-8.909, -42.569, 107.415, 170.175, 65.171, -175.841]
  MoveL 4614 to (280.7, 235.39, -10) mm, rotated rx 180 ry 0 rz 180 deg; joints [-8.975, -42.54, 107.33, 170.098, 65.119, -175.8]
  MoveL 4615 to (281.56, 237.36, -10) mm, rotated rx 180 ry 0 rz -180 deg; joints [-9.044, -42.514, 107.252, 170.018, 65.073, -175.758]
  MoveL 4616 to (282.3, 239.39, -10) mm, rotated rx -180 ry 0 rz -180 deg; joints [-9.115, -42.491, 107.181, 169.936, 65.032, -175.715]
  MoveL 4617 to (282.91, 241.46, -10) mm, rotated rx -180 ry 0 rz -180 deg; joints [-9.189, -42.47, 107.119, 169.851, 64.996, -175.673]
  MoveL 4618 to (283.39, 243.57, -10) mm, rotated rx 180 ry 0 rz -180 deg; joints [-9.265, -42.452, 107.064, 169.765, 64.967, -175.631]
  MoveL 4619 to (283.73, 245.7, -10) mm, rotated rx -180 ry 0 rz 180 deg; joints [-9.343, -42.437, 107.019, 169.677, 64.942, -175.589]
  MoveL 4620 to (283.93, 247.84, -10) mm, rotated rx -180 ry 0 rz -180 deg; joints [-9.421, -42.424, 106.981, 169.588, 64.924, -175.547]
  MoveL 4621 to (284, 250, -10) mm, rotated rx -180 ry 0 rz 180 deg; joints [-9.502, -42.415, 106.953, 169.498, 64.912, -175.506]
  MoveL 4622 to (272, 250, -10) mm, rotated rx -180 ry 0 rz 180 deg; joints [-9.577, -42.679, 107.748, 169.46, 65.44, -175.578]
  MoveL 4623 to (271.96, 251.4, -10) mm, rotated rx 180 ry 0 rz -180 deg; joints [-9.63, -42.675, 107.735, 169.401, 65.435, -175.552]
  MoveL 4624 to (271.82, 252.79, -10) mm, rotated rx 180 ry 0 rz -180 deg; joints [-9.683, -42.673, 107.728, 169.343, 65.435, -175.527]
  MoveL 4625 to (271.6, 254.16, -10) mm, rotated rx -180 ry 0 rz -180 deg; joints [-9.736, -42.672, 107.727, 169.284, 65.438, -175.502]
  MoveL 4626 to (271.29, 255.53, -10) mm, rotated rx 180 ry 0 rz 180 deg; joints [-9.789, -42.674, 107.732, 169.226, 65.446, -175.479]
  MoveL 4627 to (270.9, 256.86, -10) mm, rotated rx 180 ry 0 rz 180 deg; joints [-9.842, -42.677, 107.743, 169.169, 65.457, -175.456]
  MoveL 4628 to (270.42, 258.18, -10) mm, rotated rx 180 ry 0 rz 180 deg; joints [-9.894, -42.683, 107.759, 169.113, 65.472, -175.435]
  MoveL 4629 to (269.86, 259.46, -10) mm, rotated rx 180 ry 0 rz 180 deg; joints [-9.946, -42.69, 107.781, 169.057, 65.491, -175.414]
  MoveL 4630 to (269.22, 260.7, -10) mm, rotated rx -180 ry 0 rz -180 deg; joints [-9.997, -42.699, 107.809, 169.003, 65.513, -175.395]
  MoveL 4631 to (268.51, 261.89, -10) mm, rotated rx -180 ry 0 rz -180 deg; joints [-10.047, -42.71, 107.843, 168.951, 65.539, -175.377]
  MoveL 4632 to (267.72, 263.04, -10) mm, rotated rx -180 ry 0 rz 180 deg; joints [-10.095, -42.723, 107.881, 168.9, 65.568, -175.361]
  MoveL 4633 to (266.85, 264.14, -10) mm, rotated rx -180 ry 0 rz 180 deg; joints [-10.142, -42.737, 107.925, 168.851, 65.601, -175.346]
  MoveL 4634 to (265.92, 265.18, -10) mm, rotated rx -180 ry 0 rz -180 deg; joints [-10.188, -42.754, 107.974, 168.804, 65.637, -175.332]
  MoveL 4635 to (264.93, 266.16, -10) mm, rotated rx 180 ry 0 rz -180 deg; joints [-10.231, -42.771, 108.028, 168.76, 65.676, -175.32]
  MoveL 4636 to (263.87, 267.08, -10) mm, rotated rx -180 ry 0 rz -180 deg; joints [-10.273, -42.791, 108.087, 168.718, 65.718, -175.31]
  MoveL 4637 to (262.76, 267.92, -10) mm, rotated rx -180 ry 0 rz -180 deg; joints [-10.312, -42.811, 108.15, 168.678, 65.763, -175.301]
  MoveL 4638 to (261.6, 268.69, -10) mm, rotated rx -180 ry 0 rz -180 deg; joints [-10.35, -42.833, 108.217, 168.642, 65.81, -175.294]
  MoveL 4639 to (260.39, 269.39, -10) mm, rotated rx -180 ry 0 rz 180 deg; joints [-10.384, -42.857, 108.288, 168.608, 65.86, -175.289]
  MoveL 4640 to (259.14, 270.01, -10) mm, rotated rx -180 ry 0 rz -180 deg; joints [-10.416, -42.881, 108.363, 168.577, 65.911, -175.286]
  MoveL 4641 to (257.85, 270.55, -10) mm, rotated rx 180 ry 0 rz -180 deg; joints [-10.446, -42.907, 108.441, 168.55, 65.965, -175.284]
  MoveL 4642 to (256.53, 271.01, -10) mm, rotated rx 180 ry 0 rz -180 deg; joints [-10.472, -42.933, 108.522, 168.526, 66.021, -175.284]
  MoveL 4643 to (255.19, 271.38, -10) mm, rotated rx 180 ry 0 rz 180 deg; joints [-10.495, -42.96, 108.605, 168.505, 66.078, -175.286]
  MoveL 4644 to (253.82, 271.67, -10) mm, rotated rx 180 ry 0 rz 180 deg; joints [-10.516, -42.988, 108.691, 168.488, 66.137, -175.29]
  MoveL 4645 to (252.44, 271.86, -10) mm, rotated rx 180 ry 0 rz 180 deg; joints [-10.533, -43.017, 108.779, 168.475, 66.196, -175.295]
  MoveL 4646 to (251.05, 271.98, -10) mm, rotated rx -180 ry 0 rz -180 deg; joints [-10.547, -43.046, 108.869, 168.465, 66.257, -175.302]
  MoveL 4647 to (249.65, 272, -10) mm, rotated rx 180 ry 0 rz -180 deg; joints [-10.558, -43.075, 108.96, 168.459, 66.318, -175.311]
  MoveL 4648 to (248.26, 271.93, -10) mm, rotated rx 180 ry 0 rz 180 deg; joints [-10.565, -43.105, 109.052, 168.456, 66.379, -175.321]
  MoveL 4649 to (246.87, 271.78, -10) mm, rotated rx 180 ry 0 rz 180 deg; joints [-10.569, -43.135, 109.144, 168.457, 66.441, -175.333]
  MoveL 4650 to (245.49, 271.53, -10) mm, rotated rx 180 ry 0 rz 180 deg; joints [-10.57, -43.165, 109.237, 168.462, 66.503, -175.347]
  MoveL 4651 to (244.14, 271.2, -10) mm, rotated rx 180 ry 0 rz -180 deg; joints [-10.567, -43.195, 109.33, 168.471, 66.564, -175.362]
  MoveL 4652 to (242.8, 270.79, -10) mm, rotated rx -180 ry 0 rz -180 deg; joints [-10.56, -43.224, 109.421, 168.483, 66.624, -175.378]
  MoveL 4653 to (241.5, 270.29, -10) mm, rotated rx 180 ry 0 rz 180 deg; joints [-10.551, -43.254, 109.512, 168.499, 66.684, -175.396]
  MoveL 4654 to (240.23, 269.71, -10) mm, rotated rx 180 ry 0 rz -180 deg; joints [-10.538, -43.282, 109.602, 168.518, 66.743, -175.415]
  MoveL 4655 to (239, 269.05, -10) mm, rotated rx 180 ry 0 rz 180 deg; joints [-10.521, -43.311, 109.69, 168.541, 66.8, -175.434]
  MoveL 4656 to (237.81, 268.32, -10) mm, rotated rx -180 ry 0 rz 180 deg; joints [-10.501, -43.338, 109.776, 168.568, 66.856, -175.456]
  MoveL 4657 to (236.68, 267.51, -10) mm, rotated rx -180 ry 0 rz -180 deg; joints [-10.478, -43.365, 109.86, 168.597, 66.91, -175.478]
  MoveL 4658 to (235.59, 266.63, -10) mm, rotated rx 180 ry 0 rz 180 deg; joints [-10.452, -43.391, 109.941, 168.63, 66.962, -175.5]
  MoveL 4659 to (234.57, 265.68, -10) mm, rotated rx -180 ry 0 rz 180 deg; joints [-10.423, -43.415, 110.019, 168.666, 67.012, -175.524]
  MoveL 4660 to (233.6, 264.67, -10) mm, rotated rx -180 ry 0 rz 180 deg; joints [-10.391, -43.439, 110.094, 168.705, 67.059, -175.549]
  MoveL 4661 to (232.71, 263.6, -10) mm, rotated rx 180 ry 0 rz -180 deg; joints [-10.357, -43.462, 110.165, 168.747, 67.104, -175.573]
  MoveL 4662 to (231.88, 262.48, -10) mm, rotated rx -180 ry 0 rz 180 deg; joints [-10.319, -43.483, 110.232, 168.791, 67.146, -175.599]
  MoveL 4663 to (231.12, 261.3, -10) mm, rotated rx 180 ry 0 rz -180 deg; joints [-10.279, -43.503, 110.294, 168.838, 67.185, -175.625]
  MoveL 4664 to (230.45, 260.08, -10) mm, rotated rx 180 ry 0 rz -180 deg; joints [-10.237, -43.521, 110.353, 168.887, 67.221, -175.651]
  MoveL 4665 to (229.85, 258.82, -10) mm, rotated rx 180 ry 0 rz 180 deg; joints [-10.192, -43.538, 110.406, 168.938, 67.254, -175.677]
  MoveL 4666 to (229.33, 257.52, -10) mm, rotated rx 180 ry 0 rz -180 deg; joints [-10.146, -43.554, 110.455, 168.99, 67.283, -175.703]
  MoveL 4667 to (228.89, 256.2, -10) mm, rotated rx -180 ry 0 rz 180 deg; joints [-10.098, -43.567, 110.499, 169.045, 67.309, -175.73]
  MoveL 4668 to (228.54, 254.85, -10) mm, rotated rx 180 ry 0 rz 180 deg; joints [-10.048, -43.579, 110.537, 169.101, 67.331, -175.756]
  MoveL 4669 to (228.28, 253.48, -10) mm, rotated rx 180 ry 0 rz 180 deg; joints [-9.997, -43.59, 110.57, 169.158, 67.349, -175.782]
  MoveL 4670 to (228.1, 252.09, -10) mm, rotated rx 180 ry 0 rz -180 deg; joints [-9.945, -43.598, 110.597, 169.216, 67.364, -175.807]
  MoveL 4671 to (228.01, 250.7, -10) mm, rotated rx -180 ry 0 rz 180 deg; joints [-9.891, -43.605, 110.619, 169.274, 67.374, -175.832]
  MoveL 4672 to (228.01, 249.3, -10) mm, rotated rx -180 ry 0 rz 180 deg; joints [-9.837, -43.61, 110.634, 169.334, 67.381, -175.857]
  MoveL 4673 to (228.1, 247.91, -10) mm, rotated rx -180 ry 0 rz 180 deg; joints [-9.783, -43.613, 110.644, 169.393, 67.384, -175.881]
  MoveL 4674 to (228.28, 246.52, -10) mm, rotated rx 180 ry 0 rz -180 deg; joints [-9.728, -43.614, 110.648, 169.452, 67.382, -175.904]
  MoveL 4675 to (228.54, 245.15, -10) mm, rotated rx 180 ry 0 rz -180 deg; joints [-9.673, -43.614, 110.646, 169.512, 67.377, -175.927]
  MoveL 4676 to (228.89, 243.8, -10) mm, rotated rx -180 ry 0 rz -180 deg; joints [-9.619, -43.611, 110.638, 169.57, 67.368, -175.948]
  MoveL 4677 to (229.33, 242.48, -10) mm, rotated rx -180 ry 0 rz 180 deg; joints [-9.564, -43.607, 110.625, 169.628, 67.355, -175.969]
  MoveL 4678 to (229.85, 241.18, -10) mm, rotated rx -180 ry 0 rz 180 deg; joints [-9.511, -43.601, 110.605, 169.685, 67.338, -175.989]
  MoveL 4679 to (230.45, 239.92, -10) mm, rotated rx -180 ry 0 rz -180 deg; joints [-9.458, -43.593, 110.58, 169.741, 67.317, -176.007]
  MoveL 4680 to (231.12, 238.7, -10) mm, rotated rx -180 ry 0 rz -180 deg; joints [-9.407, -43.583, 110.549, 169.795, 67.293, -176.025]
  MoveL 4681 to (231.88, 237.52, -10) mm, rotated rx -180 ry 0 rz -180 deg; joints [-9.356, -43.572, 110.512, 169.847, 67.265, -176.041]
  MoveL 4682 to (232.71, 236.4, -10) mm, rotated rx -180 ry 0 rz 180 deg; joints [-9.308, -43.559, 110.471, 169.898, 67.233, -176.056]
  MoveL 4683 to (233.6, 235.33, -10) mm, rotated rx 180 ry 0 rz 180 deg; joints [-9.261, -43.544, 110.424, 169.947, 67.198, -176.07]
  MoveL 4684 to (234.57, 234.32, -10) mm, rotated rx 180 ry 0 rz -180 deg; joints [-9.215, -43.527, 110.372, 169.993, 67.16, -176.082]
  MoveL 4685 to (235.59, 233.37, -10) mm, rotated rx -180 ry 0 rz -180 deg; joints [-9.172, -43.509, 110.315, 170.037, 67.119, -176.093]
  MoveL 4686 to (236.68, 232.49, -10) mm, rotated rx 180 ry 0 rz -180 deg; joints [-9.132, -43.49, 110.254, 170.078, 67.075, -176.102]
  MoveL 4687 to (237.81, 231.68, -10) mm, rotated rx 180 ry 0 rz -180 deg; joints [-9.093, -43.469, 110.188, 170.116, 67.028, -176.11]
  MoveL 4688 to (239, 230.95, -10) mm, rotated rx 180 ry 0 rz 180 deg; joints [-9.058, -43.447, 110.118, 170.151, 66.979, -176.116]
  MoveL 4689 to (240.23, 230.29, -10) mm, rotated rx 180 ry 0 rz 180 deg; joints [-9.025, -43.424, 110.045, 170.183, 66.928, -176.121]
  MoveL 4690 to (241.5, 229.71, -10) mm, rotated rx 180 ry 0 rz 180 deg; joints [-8.995, -43.399, 109.968, 170.212, 66.874, -176.124]
  MoveL 4691 to (242.8, 229.21, -10) mm, rotated rx 180 ry 0 rz 180 deg; joints [-8.968, -43.374, 109.888, 170.237, 66.818, -176.125]
  MoveL 4692 to (244.14, 228.8, -10) mm, rotated rx 180 ry 0 rz -180 deg; joints [-8.943, -43.347, 109.805, 170.259, 66.761, -176.125]
  MoveL 4693 to (245.49, 228.47, -10) mm, rotated rx -180 ry 0 rz -180 deg; joints [-8.923, -43.32, 109.72, 170.278, 66.703, -176.123]
  MoveL 4694 to (246.87, 228.22, -10) mm, rotated rx 180 ry 0 rz 180 deg; joints [-8.905, -43.292, 109.633, 170.293, 66.643, -176.12]
  MoveL 4695 to (248.26, 228.07, -10) mm, rotated rx -180 ry 0 rz 180 deg; joints [-8.891, -43.264, 109.544, 170.304, 66.582, -176.115]
  MoveL 4696 to (249.65, 228, -10) mm, rotated rx -180 ry 0 rz 180 deg; joints [-8.88, -43.235, 109.453, 170.311, 66.521, -176.109]
  MoveL 4697 to (251.05, 228.02, -10) mm, rotated rx -180 ry 0 rz -180 deg; joints [-8.872, -43.205, 109.361, 170.315, 66.459, -176.1]
  MoveL 4698 to (252.44, 228.14, -10) mm, rotated rx -180 ry 0 rz 180 deg; joints [-8.868, -43.175, 109.269, 170.315, 66.397, -176.091]
  MoveL 4699 to (253.82, 228.33, -10) mm, rotated rx 180 ry 0 rz 180 deg; joints [-8.868, -43.145, 109.176, 170.311, 66.335, -176.079]
  MoveL 4700 to (255.19, 228.62, -10) mm, rotated rx 180 ry 0 rz 180 deg; joints [-8.87, -43.116, 109.084, 170.303, 66.273, -176.067]
  MoveL 4701 to (256.53, 228.99, -10) mm, rotated rx -180 ry 0 rz -180 deg; joints [-8.877, -43.086, 108.992, 170.292, 66.212, -176.053]
  MoveL 4702 to (257.85, 229.45, -10) mm, rotated rx 180 ry 0 rz 180 deg; joints [-8.886, -43.056, 108.9, 170.277, 66.152, -176.037]
  MoveL 4703 to (259.14, 229.99, -10) mm, rotated rx 180 ry 0 rz -180 deg; joints [-8.899, -43.027, 108.81, 170.258, 66.093, -176.02]
  MoveL 4704 to (260.39, 230.61, -10) mm, rotated rx -180 ry 0 rz 180 deg; joints [-8.915, -42.998, 108.721, 170.236, 66.035, -176.002]
  MoveL 4705 to (261.6, 231.31, -10) mm, rotated rx -180 ry 0 rz 180 deg; joints [-8.934, -42.97, 108.635, 170.21, 65.979, -175.982]
  MoveL 4706 to (262.76, 232.08, -10) mm, rotated rx 180 ry 0 rz -180 deg; joints [-8.957, -42.942, 108.55, 170.182, 65.924, -175.962]
  MoveL 4707 to (263.87, 232.92, -10) mm, rotated rx 180 ry 0 rz -180 deg; joints [-8.982, -42.916, 108.468, 170.15, 65.872, -175.94]
  MoveL 4708 to (264.93, 233.84, -10) mm, rotated rx 180 ry 0 rz -180 deg; joints [-9.011, -42.89, 108.389, 170.115, 65.821, -175.917]
  MoveL 4709 to (265.92, 234.82, -10) mm, rotated rx -180 ry 0 rz -180 deg; joints [-9.042, -42.865, 108.313, 170.077, 65.773, -175.894]
  MoveL 4710 to (266.85, 235.86, -10) mm, rotated rx 180 ry 0 rz 180 deg; joints [-9.076, -42.841, 108.241, 170.036, 65.728, -175.869]
  MoveL 4711 to (267.72, 236.96, -10) mm, rotated rx -180 ry 0 rz -180 deg; joints [-9.112, -42.819, 108.172, 169.993, 65.685, -175.844]
  MoveL 4712 to (268.51, 238.11, -10) mm, rotated rx -180 ry 0 rz 180 deg; joints [-9.15, -42.798, 108.108, 169.947, 65.645, -175.819]
  MoveL 4713 to (269.22, 239.3, -10) mm, rotated rx 180 ry 0 rz 180 deg; joints [-9.191, -42.778, 108.048, 169.899, 65.608, -175.792]
  MoveL 4714 to (269.86, 240.54, -10) mm, rotated rx 180 ry 0 rz 180 deg; joints [-9.234, -42.76, 107.992, 169.849, 65.575, -175.766]
  MoveL 4715 to (270.42, 241.82, -10) mm, rotated rx 180 ry 0 rz -180 deg; joints [-9.279, -42.743, 107.942, 169.797, 65.545, -175.739]
  MoveL 4716 to (270.9, 243.14, -10) mm, rotated rx 180 ry 0 rz -180 deg; joints [-9.326, -42.728, 107.896, 169.744, 65.518, -175.712]
  MoveL 4717 to (271.29, 244.47, -10) mm, rotated rx 180 ry 0 rz 180 deg; joints [-9.374, -42.714, 107.855, 169.689, 65.495, -175.685]
  MoveL 4718 to (271.6, 245.84, -10) mm, rotated rx -180 ry 0 rz -180 deg; joints [-9.423, -42.703, 107.82, 169.633, 65.475, -175.658]
  MoveL 4719 to (271.82, 247.22, -10) mm, rotated rx 180 ry 0 rz -180 deg; joints [-9.473, -42.693, 107.79, 169.576, 65.46, -175.631]
  MoveL 4720 to (271.96, 248.6, -10) mm, rotated rx 180 ry 0 rz -180 deg; joints [-9.525, -42.685, 107.766, 169.518, 65.448, -175.604]
  MoveL 4721 to (272, 250, -10) mm, rotated rx -180 ry 0 rz 180 deg; joints [-9.577, -42.679, 107.748, 169.46, 65.44, -175.578]
  MoveL 4722 to (260, 250, -10) mm, rotated rx 180 ry 0 rz 180 deg; joints [-9.654, -42.939, 108.539, 169.42, 65.968, -175.65]
  MoveL 4723 to (259.98, 250.63, -10) mm, rotated rx 180 ry 0 rz 180 deg; joints [-9.678, -42.937, 108.533, 169.393, 65.966, -175.638]
  MoveL 4724 to (259.92, 251.27, -10) mm, rotated rx -180 ry 0 rz -180 deg; joints [-9.702, -42.936, 108.53, 169.366, 65.965, -175.627]
  MoveL 4725 to (259.82, 251.89, -10) mm, rotated rx -180 ry 0 rz -180 deg; joints [-9.727, -42.935, 108.529, 169.34, 65.967, -175.616]
  MoveL 4726 to (259.68, 252.51, -10) mm, rotated rx -180 ry 0 rz 180 deg; joints [-9.751, -42.936, 108.531, 169.313, 65.97, -175.606]
  MoveL 4727 to (259.5, 253.12, -10) mm, rotated rx -180 ry 0 rz 180 deg; joints [-9.775, -42.938, 108.536, 169.287, 65.975, -175.596]
  MoveL 4728 to (259.28, 253.72, -10) mm, rotated rx 180 ry 0 rz -180 deg; joints [-9.799, -42.94, 108.544, 169.261, 65.982, -175.586]
  MoveL 4729 to (259.03, 254.3, -10) mm, rotated rx 180 ry 0 rz -180 deg; joints [-9.823, -42.944, 108.554, 169.236, 65.991, -175.577]
  MoveL 4730 to (258.74, 254.86, -10) mm, rotated rx 180 ry 0 rz 180 deg; joints [-9.846, -42.948, 108.567, 169.211, 66.001, -175.568]
  MoveL 4731 to (258.41, 255.41, -10) mm, rotated rx 180 ry 0 rz -180 deg; joints [-9.869, -42.953, 108.582, 169.187, 66.013, -175.56]
  MoveL 4732 to (258.05, 255.93, -10) mm, rotated rx -180 ry 0 rz 180 deg; joints [-9.891, -42.958, 108.599, 169.164, 66.026, -175.553]
  MoveL 4733 to (257.66, 256.43, -10) mm, rotated rx 180 ry 0 rz -180 deg; joints [-9.913, -42.965, 108.619, 169.142, 66.041, -175.546]
  MoveL 4734 to (257.24, 256.9, -10) mm, rotated rx 180 ry 0 rz 180 deg; joints [-9.933, -42.972, 108.642, 169.121, 66.057, -175.54]
  MoveL 4735 to (256.79, 257.35, -10) mm, rotated rx -180 ry 0 rz 180 deg; joints [-9.953, -42.98, 108.666, 169.1, 66.075, -175.535]
  MoveL 4736 to (256.31, 257.76, -10) mm, rotated rx 180 ry 0 rz 180 deg; joints [-9.972, -42.989, 108.693, 169.081, 66.094, -175.53]
  MoveL 4737 to (255.8, 258.15, -10) mm, rotated rx -180 ry 0 rz -180 deg; joints [-9.99, -42.998, 108.722, 169.063, 66.115, -175.526]
  MoveL 4738 to (255.27, 258.5, -10) mm, rotated rx -180 ry 0 rz -180 deg; joints [-10.007, -43.008, 108.752, 169.047, 66.136, -175.523]
  MoveL 4739 to (254.72, 258.81, -10) mm, rotated rx -180 ry 0 rz 180 deg; joints [-10.023, -43.019, 108.785, 169.031, 66.159, -175.521]
  MoveL 4740 to (254.15, 259.1, -10) mm, rotated rx -180 ry 0 rz -180 deg; joints [-10.037, -43.03, 108.819, 169.017, 66.183, -175.519]
  MoveL 4741 to (253.57, 259.34, -10) mm, rotated rx 180 ry 0 rz 180 deg; joints [-10.05, -43.041, 108.854, 169.005, 66.207, -175.518]
  MoveL 4742 to (252.97, 259.55, -10) mm, rotated rx 180 ry 0 rz -180 deg; joints [-10.062, -43.053, 108.891, 168.994, 66.233, -175.518]
  MoveL 4743 to (252.36, 259.72, -10) mm, rotated rx -180 ry 0 rz -180 deg; joints [-10.073, -43.065, 108.929, 168.985, 66.259, -175.519]
  MoveL 4744 to (251.74, 259.85, -10) mm, rotated rx 180 ry 0 rz -180 deg; joints [-10.082, -43.078, 108.968, 168.977, 66.285, -175.52]
  MoveL 4745 to (251.11, 259.94, -10) mm, rotated rx -180 ry 0 rz 180 deg; joints [-10.09, -43.091, 109.008, 168.971, 66.313, -175.523]
  MoveL 4746 to (250.48, 259.99, -10) mm, rotated rx -180 ry 0 rz -180 deg; joints [-10.096, -43.104, 109.049, 168.967, 66.34, -175.526]
  MoveL 4747 to (249.84, 260, -10) mm, rotated rx -180 ry 0 rz 180 deg; joints [-10.101, -43.118, 109.091, 168.964, 66.368, -175.53]
  MoveL 4748 to (249.21, 259.97, -10) mm, rotated rx -180 ry 0 rz -180 deg; joints [-10.104, -43.131, 109.132, 168.963, 66.396, -175.534]
  MoveL 4749 to (248.58, 259.9, -10) mm, rotated rx 180 ry 0 rz -180 deg; joints [-10.105, -43.145, 109.174, 168.963, 66.424, -175.539]
  MoveL 4750 to (247.95, 259.79, -10) mm, rotated rx 180 ry 0 rz -180 deg; joints [-10.105, -43.158, 109.216, 168.966, 66.452, -175.545]
  MoveL 4751 to (247.34, 259.64, -10) mm, rotated rx 180 ry 0 rz -180 deg; joints [-10.104, -43.172, 109.259, 168.97, 66.48, -175.552]
  MoveL 4752 to (246.73, 259.45, -10) mm, rotated rx -180 ry 0 rz -180 deg; joints [-10.101, -43.185, 109.3, 168.975, 66.508, -175.559]
  MoveL 4753 to (246.14, 259.22, -10) mm, rotated rx -180 ry 0 rz -180 deg; joints [-10.096, -43.199, 109.342, 168.983, 66.535, -175.567]
  MoveL 4754 to (245.56, 258.96, -10) mm, rotated rx 180 ry 0 rz -180 deg; joints [-10.09, -43.212, 109.382, 168.992, 66.561, -175.575]
  MoveL 4755 to (245, 258.66, -10) mm, rotated rx -180 ry 0 rz 180 deg; joints [-10.082, -43.225, 109.422, 169.002, 66.587, -175.584]
  MoveL 4756 to (244.46, 258.33, -10) mm, rotated rx 180 ry 0 rz 180 deg; joints [-10.073, -43.237, 109.461, 169.014, 66.613, -175.594]
  MoveL 4757 to (243.94, 257.96, -10) mm, rotated rx -180 ry 0 rz -180 deg; joints [-10.063, -43.249, 109.499, 169.028, 66.637, -175.604]
  MoveL 4758 to (243.45, 257.56, -10) mm, rotated rx 180 ry 0 rz 180 deg; joints [-10.051, -43.261, 109.536, 169.043, 66.661, -175.614]
  MoveL 4759 to (242.99, 257.13, -10) mm, rotated rx -180 ry 0 rz -180 deg; joints [-10.037, -43.273, 109.572, 169.059, 66.683, -175.625]
  MoveL 4760 to (242.55, 256.67, -10) mm, rotated rx -180 ry 0 rz -180 deg; joints [-10.023, -43.283, 109.605, 169.077, 66.705, -175.636]
  MoveL 4761 to (242.14, 256.18, -10) mm, rotated rx 180 ry 0 rz -180 deg; joints [-10.007, -43.294, 109.638, 169.096, 66.725, -175.647]
  MoveL 4762 to (241.76, 255.67, -10) mm, rotated rx 180 ry 0 rz -180 deg; joints [-9.99, -43.303, 109.668, 169.116, 66.744, -175.659]
  MoveL 4763 to (241.42, 255.14, -10) mm, rotated rx 180 ry 0 rz 180 deg; joints [-9.972, -43.313, 109.696, 169.137, 66.762, -175.67]
  MoveL 4764 to (241.11, 254.58, -10) mm, rotated rx 180 ry 0 rz 180 deg; joints [-9.953, -43.321, 109.723, 169.16, 66.778, -175.682]
  MoveL 4765 to (240.84, 254.01, -10) mm, rotated rx -180 ry 0 rz 180 deg; joints [-9.933, -43.329, 109.747, 169.183, 66.793, -175.694]
  MoveL 4766 to (240.6, 253.42, -10) mm, rotated rx -180 ry 0 rz 180 deg; joints [-9.912, -43.336, 109.769, 169.207, 66.806, -175.706]
  MoveL 4767 to (240.41, 252.82, -10) mm, rotated rx 180 ry 0 rz 180 deg; joints [-9.89, -43.342, 109.789, 169.232, 66.818, -175.718]
  MoveL 4768 to (240.25, 252.2, -10) mm, rotated rx -180 ry 0 rz -180 deg; joints [-9.867, -43.348, 109.806, 169.257, 66.827, -175.73]
  MoveL 4769 to (240.13, 251.58, -10) mm, rotated rx -180 ry 0 rz 180 deg; joints [-9.844, -43.352, 109.821, 169.283, 66.836, -175.742]
  MoveL 4770 to (240.05, 250.95, -10) mm, rotated rx -180 ry 0 rz -180 deg; joints [-9.821, -43.356, 109.834, 169.309, 66.842, -175.754]
  MoveL 4771 to (240, 250.32, -10) mm, rotated rx -180 ry 0 rz -180 deg; joints [-9.797, -43.36, 109.843, 169.336, 66.847, -175.766]
  MoveL 4772 to (240, 249.68, -10) mm, rotated rx -180 ry 0 rz -180 deg; joints [-9.772, -43.362, 109.851, 169.362, 66.85, -175.777]
  MoveL 4773 to (240.05, 249.05, -10) mm, rotated rx 180 ry 0 rz -180 deg; joints [-9.748, -43.363, 109.855, 169.389, 66.851, -175.788]
  MoveL 4774 to (240.13, 248.42, -10) mm, rotated rx -180 ry 0 rz 180 deg; joints [-9.723, -43.364, 109.857, 169.416, 66.85, -175.799]
  MoveL 4775 to (240.25, 247.8, -10) mm, rotated rx 180 ry 0 rz -180 deg; joints [-9.698, -43.364, 109.856, 169.443, 66.848, -175.809]
  MoveL 4776 to (240.41, 247.18, -10) mm, rotated rx 180 ry 0 rz 180 deg; joints [-9.674, -43.362, 109.852, 169.47, 66.844, -175.819]
  MoveL 4777 to (240.6, 246.58, -10) mm, rotated rx -180 ry 0 rz 180 deg; joints [-9.649, -43.36, 109.846, 169.496, 66.838, -175.829]
  MoveL 4778 to (240.84, 245.99, -10) mm, rotated rx 180 ry 0 rz -180 deg; joints [-9.625, -43.358, 109.837, 169.521, 66.83, -175.838]
  MoveL 4779 to (241.11, 245.42, -10) mm, rotated rx 180 ry 0 rz 180 deg; joints [-9.601, -43.354, 109.826, 169.547, 66.821, -175.847]
  MoveL 4780 to (241.42, 244.86, -10) mm, rotated rx -180 ry 0 rz 180 deg; joints [-9.578, -43.349, 109.812, 169.571, 66.81, -175.855]
  MoveL 4781 to (241.76, 244.33, -10) mm, rotated rx 180 ry 0 rz 180 deg; joints [-9.555, -43.344, 109.795, 169.595, 66.797, -175.862]
  MoveL 4782 to (242.14, 243.82, -10) mm, rotated rx -180 ry 0 rz 180 deg; joints [-9.533, -43.338, 109.776, 169.618, 66.783, -175.869]
  MoveL 4783 to (242.55, 243.33, -10) mm, rotated rx -180 ry 0 rz 180 deg; joints [-9.512, -43.331, 109.755, 169.64, 66.767, -175.875]
  MoveL 4784 to (242.99, 242.87, -10) mm, rotated rx -180 ry 0 rz -180 deg; joints [-9.491, -43.324, 109.732, 169.661, 66.75, -175.881]
  MoveL 4785 to (243.45, 242.44, -10) mm, rotated rx -180 ry 0 rz 180 deg; joints [-9.472, -43.316, 109.706, 169.681, 66.731, -175.886]
  MoveL 4786 to (243.94, 242.04, -10) mm, rotated rx 180 ry 0 rz 180 deg; joints [-9.453, -43.307, 109.678, 169.699, 66.711, -175.89]
  MoveL 4787 to (244.46, 241.67, -10) mm, rotated rx 180 ry 0 rz 180 deg; joints [-9.436, -43.297, 109.648, 169.717, 66.69, -175.894]
  MoveL 4788 to (245, 241.34, -10) mm, rotated rx -180 ry 0 rz 180 deg; joints [-9.42, -43.287, 109.617, 169.733, 66.668, -175.896]
  MoveL 4789 to (245.56, 241.04, -10) mm, rotated rx 180 ry 0 rz -180 deg; joints [-9.405, -43.276, 109.583, 169.747, 66.645, -175.899]
  MoveL 4790 to (246.14, 240.78, -10) mm, rotated rx -180 ry 0 rz 180 deg; joints [-9.391, -43.265, 109.549, 169.76, 66.62, -175.9]
  MoveL 4791 to (246.73, 240.55, -10) mm, rotated rx -180 ry 0 rz -180 deg; joints [-9.379, -43.254, 109.512, 169.772, 66.595, -175.9]
  MoveL 4792 to (247.34, 240.36, -10) mm, rotated rx 180 ry 0 rz 180 deg; joints [-9.368, -43.242, 109.475, 169.782, 66.569, -175.9]
  MoveL 4793 to (247.95, 240.21, -10) mm, rotated rx -180 ry 0 rz -180 deg; joints [-9.358, -43.229, 109.436, 169.79, 66.543, -175.899]
  MoveL 4794 to (248.58, 240.1, -10) mm, rotated rx -180 ry 0 rz 180 deg; joints [-9.35, -43.216, 109.396, 169.797, 66.516, -175.898]
  MoveL 4795 to (249.21, 240.03, -10) mm, rotated rx -180 ry 0 rz 180 deg; joints [-9.343, -43.203, 109.356, 169.802, 66.488, -175.895]
  MoveL 4796 to (249.84, 240, -10) mm, rotated rx -180 ry 0 rz 180 deg; joints [-9.338, -43.19, 109.315, 169.806, 66.46, -175.892]
  MoveL 4797 to (250.48, 240.01, -10) mm, rotated rx -180 ry 0 rz -180 deg; joints [-9.334, -43.177, 109.273, 169.808, 66.432, -175.888]
  MoveL 4798 to (251.11, 240.06, -10) mm, rotated rx -180 ry 0 rz -180 deg; joints [-9.332, -43.163, 109.231, 169.808, 66.404, -175.884]
  MoveL 4799 to (251.74, 240.15, -10) mm, rotated rx 180 ry 0 rz 180 deg; joints [-9.332, -43.15, 109.189, 169.806, 66.376, -175.878]
  MoveL 4800 to (252.36, 240.28, -10) mm, rotated rx 180 ry 0 rz 180 deg; joints [-9.333, -43.136, 109.147, 169.803, 66.348, -175.872]
  MoveL 4801 to (252.97, 240.45, -10) mm, rotated rx -180 ry 0 rz -180 deg; joints [-9.335, -43.122, 109.105, 169.797, 66.32, -175.866]
  MoveL 4802 to (253.57, 240.66, -10) mm, rotated rx 180 ry 0 rz -180 deg; joints [-9.34, -43.109, 109.063, 169.791, 66.293, -175.858]
  MoveL 4803 to (254.15, 240.9, -10) mm, rotated rx -180 ry 0 rz 180 deg; joints [-9.345, -43.096, 109.022, 169.782, 66.266, -175.851]
  MoveL 4804 to (254.72, 241.19, -10) mm, rotated rx 180 ry 0 rz 180 deg; joints [-9.352, -43.083, 108.982, 169.772, 66.24, -175.842]
  MoveL 4805 to (255.27, 241.5, -10) mm, rotated rx -180 ry 0 rz 180 deg; joints [-9.361, -43.07, 108.943, 169.761, 66.214, -175.833]
  MoveL 4806 to (255.8, 241.85, -10) mm, rotated rx 180 ry 0 rz 180 deg; joints [-9.371, -43.057, 108.904, 169.748, 66.189, -175.824]
  MoveL 4807 to (256.31, 242.24, -10) mm, rotated rx 180 ry 0 rz 180 deg; joints [-9.383, -43.045, 108.867, 169.734, 66.165, -175.814]
  MoveL 4808 to (256.79, 242.65, -10) mm, rotated rx 180 ry 0 rz 180 deg; joints [-9.395, -43.034, 108.831, 169.718, 66.142, -175.803]
  MoveL 4809 to (257.24, 243.1, -10) mm, rotated rx 180 ry 0 rz -180 deg; joints [-9.409, -43.022, 108.796, 169.7, 66.12, -175.793]
  MoveL 4810 to (257.66, 243.57, -10) mm, rotated rx -180 ry 0 rz 180 deg; joints [-9.425, -43.012, 108.763, 169.682, 66.1, -175.782]
  MoveL 4811 to (258.05, 244.07, -10) mm, rotated rx 180 ry 0 rz 180 deg; joints [-9.441, -43.002, 108.732, 169.662, 66.08, -175.77]
  MoveL 4812 to (258.41, 244.59, -10) mm, rotated rx -180 ry 0 rz -180 deg; joints [-9.459, -42.992, 108.703, 169.642, 66.062, -175.758]
  MoveL 4813 to (258.74, 245.14, -10) mm, rotated rx 180 ry 0 rz -180 deg; joints [-9.477, -42.983, 108.675, 169.62, 66.045, -175.747]
  MoveL 4814 to (259.03, 245.7, -10) mm, rotated rx 180 ry 0 rz -180 deg; joints [-9.497, -42.975, 108.65, 169.597, 66.03, -175.735]
  MoveL 4815 to (259.28, 246.28, -10) mm, rotated rx 180 ry 0 rz 180 deg; joints [-9.517, -42.967, 108.627, 169.574, 66.016, -175.722]
  MoveL 4816 to (259.5, 246.88, -10) mm, rotated rx 180 ry 0 rz 180 deg; joints [-9.539, -42.961, 108.606, 169.549, 66.004, -175.71]
  MoveL 4817 to (259.68, 247.49, -10) mm, rotated rx 180 ry 0 rz -180 deg; joints [-9.561, -42.955, 108.588, 169.524, 65.993, -175.698]
  MoveL 4818 to (259.82, 248.11, -10) mm, rotated rx -180 ry 0 rz 180 deg; joints [-9.583, -42.949, 108.572, 169.499, 65.984, -175.686]
  MoveL 4819 to (259.92, 248.73, -10) mm, rotated rx 180 ry 0 rz -180 deg; joints [-9.606, -42.945, 108.558, 169.473, 65.977, -175.674]
  MoveL 4820 to (259.98, 249.37, -10) mm, rotated rx -180 ry 0 rz -180 deg; joints [-9.63, -42.941, 108.547, 169.446, 65.971, -175.662]
  MoveL 4821 to (260, 250, -10) mm, rotated rx 180 ry 0 rz 180 deg; joints [-9.654, -42.939, 108.539, 169.42, 65.968, -175.65]
  Establecer velocidad (1000.0 mm/s)
  MoveL 4822 to (260, 250, 10) mm, rotated rx 180 ry 0 rz -180 deg; joints [-9.654, -44.022, 108.777, 169.349, 65.137, -175.479]
  MoveL 4823 to (392, 250, 10) mm, rotated rx -180 ry 0 rz -180 deg; joints [-8.871, -40.818, 99.818, 169.68, 59.411, -174.706]
  MoveL 4824 to (392, 250, 10) mm, rotated rx -180 ry 0 rz -180 deg; joints [-8.871, -40.818, 99.818, 169.68, 59.411, -174.706]
  MoveL 4825 to (392, 250, 110) mm, rotated rx 180 ry 0 rz -180 deg; joints [-8.871, -45.644, 100.623, 169.209, 55.458, -173.832]

--- program Machining2 (robot KUKA KR 200 comp) ---
  Suave(1)
  Llamar SetRPM(3000.0)
  Llamar M_RunCode(3)
  Establecer velocidad (1000.0 mm/s)
  Est. Ref.: MECANIZADO
  Est. herr: Teknomotor ATC710039 Spindle
  Mostrar Teknomotor ATC710039 Spindle
  MoveJ 1 to (75, 75, 300) mm, rotated rx -180 ry 0 rz 180 deg; joints [-3.341, -65.898, 122.818, 176.014, 56.983, -177.826]
  MoveL 2 to (75, 75, 300) mm, rotated rx -180 ry 0 rz 180 deg; joints [-3.341, -65.898, 122.818, 176.014, 56.983, -177.826]
  MoveL 3 to (75, 75, 200) mm, rotated rx 180 ry 0 rz -180 deg; joints [-3.341, -59.94, 123.126, 176.257, 63.235, -178.313]
  MoveL 4 to (75, 75, 200) mm, rotated rx 180 ry 0 rz -180 deg; joints [-3.341, -59.94, 123.126, 176.257, 63.235, -178.313]
  Establecer velocidad (1000.0 mm/s)
  MoveL 5 to (75, 75, 200) mm, rotated rx 180 ry 0 rz -180 deg; joints [-3.341, -59.94, 123.126, 176.257, 63.235, -178.313]
  MoveL 6 to (75, 75, 5) mm, rotated rx 180 ry 0 rz -180 deg; joints [-3.341, -47.608, 121.808, 176.528, 74.228, -179.055]
  Establecer velocidad (4.2 mm/s)
  MoveL 7 to (75, 75, -50) mm, rotated rx -180 ry 0 rz -180 deg; joints [-3.341, -44.065, 120.989, 176.57, 76.947, -179.224]
  Establecer velocidad (8.3 mm/s)
  MoveL 8 to (75, 75, 5) mm, rotated rx 180 ry 0 rz -180 deg; joints [-3.341, -47.608, 121.808, 176.528, 74.228, -179.055]
  Establecer velocidad (1000.0 mm/s)
  MoveL 9 to (425, 75, 5) mm, rotated rx -180 ry 0 rz -180 deg; joints [-2.627, -40.164, 98.672, 176.92, 58.545, -178.392]
  Establecer velocidad (4.2 mm/s)
  MoveL 10 to (425, 75, -50) mm, rotated rx 180 ry 0 rz 180 deg; joints [-2.627, -37.463, 97.98, 176.983, 60.552, -178.516]
  Establecer velocidad (8.3 mm/s)
  MoveL 11 to (425, 75, 5) mm, rotated rx -180 ry 0 rz -180 deg; joints [-2.627, -40.164, 98.672, 176.92, 58.545, -178.392]
  Establecer velocidad (1000.0 mm/s)
  MoveL 12 to (425, 425, 5) mm, rotated rx -180 ry 0 rz -180 deg; joints [-14.573, -38.704, 94.855, 162.617, 57.378, -170.421]
  Establecer velocidad (4.2 mm/s)
  MoveL 13 to (425, 425, -50) mm, rotated rx -180 ry 0 rz 180 deg; joints [-14.573, -36.093, 94.17, 162.97, 59.219, -171.091]
  Establecer velocidad (8.3 mm/s)
  MoveL 14 to (425, 425, 5) mm, rotated rx -180 ry 0 rz -180 deg; joints [-14.573, -38.704, 94.855, 162.617, 57.378, -170.421]
  Establecer velocidad (1000.0 mm/s)
  MoveL 15 to (75, 425, 5) mm, rotated rx -180 ry 0 rz -180 deg; joints [-18.305, -46.518, 117.66, 160.731, 72.129, -173.877]
  Establecer velocidad (4.2 mm/s)
  MoveL 16 to (75, 425, -50) mm, rotated rx -180 ry 0 rz 180 deg; joints [-18.305, -43.175, 116.877, 160.983, 74.548, -174.753]
  Establecer velocidad (8.3 mm/s)
  MoveL 17 to (75, 425, 5) mm, rotated rx -180 ry 0 rz -180 deg; joints [-18.305, -46.518, 117.66, 160.731, 72.129, -173.877]
  Establecer velocidad (1000.0 mm/s)
  MoveL 18 to (75, 425, 200) mm, rotated rx -180 ry 0 rz 180 deg; joints [-18.305, -58.076, 118.917, 159.252, 62.446, -170.06]
  MoveL 19 to (75, 425, 200) mm, rotated rx -180 ry 0 rz 180 deg; joints [-18.305, -58.076, 118.917, 159.252, 62.446, -170.06]
  MoveL 20 to (75, 425, 300) mm, rotated rx 180 ry 0 rz -180 deg; joints [-18.305, -63.639, 118.623, 158.005, 56.991, -167.59]
